(* IEC 61131-3 sources: stil/testdata, 3 files *)

(* ---- class_method.st ---- *)
CLASS MyClass
    VAR
        x, y : INT;
        temperature: REAL := 38.2;
    END_VAR

    METHOD testMethod
        VAR_INPUT myMethodArg : INT; END_VAR
        VAR myMethodLocalVar : INT; END_VAR

        x := myMethodArg;
        y := 2
    END_METHOD
END_CLASS

(* ---- basic.st ---- *)
VAR
    a, b, c: INT := 10;
    s: STRING;
    d: REAL := 9.6;
END_VAR

(* ---- simple_program.st ---- *)
PROGRAM main_prg
    VAR
        a, b, c: INT := 10;
        s: STRING;
        d: REAL := 9.6;
    END_VAR
END_PROGRAM

ACTION some_action
    a := 91;
END_ACTION
